PROGRAM main
VAR
	Blink_Status : bool;
	PB1 AT %IX0.0 : bool;
	Blink_Timer1 : TON;
	Blink_Timer2 : TOF;
	Wait_Time : time := T#2s;
	LED1 AT %QX0.0 : bool;
	TON0 : TON;
	TOF0 : TOF;
END_VAR

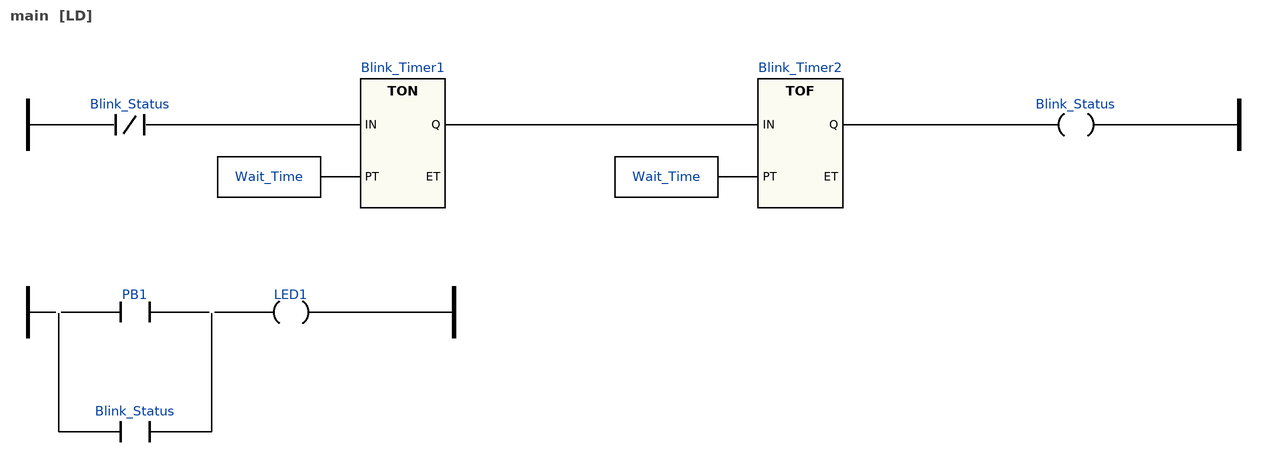
(* LD diagram, written out as Structured Text *)
Blink_Timer1(IN := NOT Blink_Status, PT := Wait_Time);
Blink_Timer2(IN := Blink_Timer1.Q, PT := Wait_Time);
Blink_Status := Blink_Timer2.Q;
LED1 := PB1 OR Blink_Status;
END_PROGRAM
